FUNCTION_BLOCK EL4032
VAR
	_io : EL4xx2_Data;
	{attribute addProperty Name "WcState"}
	_wcState : WcStateBase;
	{attribute addProperty Name "Info data"}
	_infoData : InfoDataAds;
END_VAR

PROPERTY IO : REFERENCE TO EL4xx2_Data
GET
IO REF= _io;
END_GET
END_PROPERTY

PROPERTY WcState : REFERENCE TO WcStateBase
GET
WcState REF= _wcState;
END_GET
END_PROPERTY

END_FUNCTION_BLOCK

(* stored: Version 1.1.0.1, ProductVersion 3.1.4024.9
   POU EL4032: Id {8c84147a-2426-0319-0933-6e3cee205e24}, SpecialFunc None
   Property IO: Id {bce5c38e-48fb-003e-10f5-3575d54ba771}
   Get Get: Id {d94c0e2c-e4a0-07f4-0595-1a86030981be}
   Property WcState: Id {b91aeec0-7850-0bac-0afd-f7279a6b22cf}
   Get Get: Id {4b0d50e4-62ff-0d95-20ea-35d923cb9ac6} *)
